# EPICS SNL sequencer program: pauApp/src/sncPau.stt
/*
 *    sncPau.stt
 *    Auth: KHKIM
 *
*/

program sncPau
option +r;

%{
#define ADMIN_OFF         0
#define ADMIN_ON          1
#define ADMIN_UNAVAILABLE 2
#define FBCK_OFF          0
#define FBCK_ON           1
}%

int       index;

int       feedback_mode;
assign    feedback_mode  to "{MUX_NAME}:FBCK";
monitor   feedback_mode;

double    offset[4];
assign    offset         to { "{MUX_NAME}:OFFSET_0",
                              "{MUX_NAME}:OFFSET_1",
                              "{MUX_NAME}:OFFSET_2",
                              "{MUX_NAME}:OFFSET_3" };
double    fcom[4];
assign    fcom          to { "{MUX_NAME}:GETFCOM_0",
                             "{MUX_NAME}:GETFCOM_1",
                             "{MUX_NAME}:GETFCOM_2",
                             "{MUX_NAME}:GETFCOM_3" };
monitor   fcom;

evflag    ev_fcom_0;
evflag    ev_fcom_1;
evflag    ev_fcom_2;
evflag    ev_fcom_3;

sync      fcom[0]   ev_fcom_0;
sync      fcom[1]   ev_fcom_1;
sync      fcom[2]   ev_fcom_2;
sync      fcom[3]   ev_fcom_3;

double    master;
assign    master        to "{MUX_NAME}";

int       admin;
assign    admin   to  "{ADMIN_NAME}";
monitor   admin;
evflag    ev_admin;
sync      admin    ev_admin;

ss bwProp
{
    state calc_bwProp
    {
        when(feedback_mode && efTestAndClear(ev_fcom_0)) {
            master = fcom[0];
            offset[0] = fcom[0] - master;
            pvPut(offset[0]);
            pvPut(master);
        } state calc_bwProp

        when(feedback_mode && efTestAndClear(ev_fcom_1)) {
            master = fcom[0];
            offset[1] = fcom[1] - master;
            pvPut(offset[1]);
            pvPut(master);
        } state calc_bwProp

        when(feedback_mode && efTestAndClear(ev_fcom_2)) {
            master = fcom[0];
            offset[2] = fcom[2] - master;
            pvPut(offset[2]);
            pvPut(master);
        } state calc_bwProp

        when(feedback_mode && efTestAndClear(ev_fcom_3)) {
            master = fcom[0];
            offset[3] = fcom[3] - master;
            pvPut(offset[3]);
            pvPut(master);
        } state calc_bwProp
    }

}

ss iocAdmin
{
    state init
    {
        when(admin == ADMIN_UNAVAILABLE) {
            admin = ADMIN_OFF;
            pvPut(admin);
        } state check_mode

       when(1) {
       } state check_mode
    }

    state check_mode
    {
        when(1) {
            if(admin == ADMIN_OFF)         { feedback_mode = FBCK_OFF; pvPut(feedback_mode); }
            if(admin == ADMIN_ON)          { feedback_mode = FBCK_ON;  pvPut(feedback_mode); }
            if(admin == ADMIN_UNAVAILABLE) { feedback_mode = FBCK_OFF; pvPut(feedback_mode); }
        } state wait_admin
    }

    state wait_admin
    {
        when(efTestAndClear(ev_admin)) {
        } state check_mode
    }
}
